FUNCTION F_LogL4 
VAR_INPUT
	eLogLevel		: E_LogLevel;
	sLogger			: T_MaxString;
	sMessage		: T_MaxString;
	stArg1			: T_Arg;
	stArg2			: T_Arg;
	stArg3			: T_Arg;
	stArg4			: T_Arg;
END_VAR

F_LogTArg(
	eLogLevel, 
	sLogger, 
	sMessage, 
	stArg1, 
	stArg2, 
	stArg3, 
	stArg4, 
	Tc2_Utilities.EMPTY_ARG_VALUE, 
	Tc2_Utilities.EMPTY_ARG_VALUE, 
	Tc2_Utilities.EMPTY_ARG_VALUE, 
	Tc2_Utilities.EMPTY_ARG_VALUE, 
	Tc2_Utilities.EMPTY_ARG_VALUE, 
	Tc2_Utilities.EMPTY_ARG_VALUE, 
	0
);

END_FUNCTION

(* stored: Version 1.1.0.1, ProductVersion 3.1.4024.0
   POU F_LogL4: Id {6a47f052-06c1-4b71-952d-4cf0826a3337}, SpecialFunc None *)
